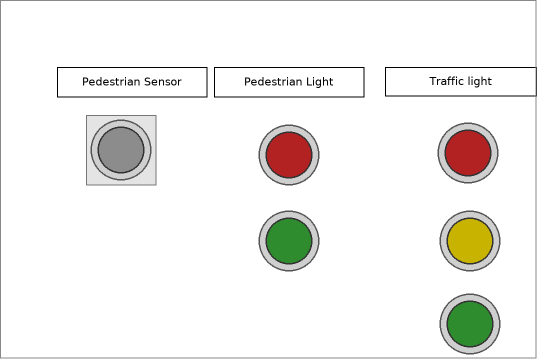
VISUALIZATION Visualization_Trafficlight  // 537x359
    Lamp1 (433,118 70x70), variable: GVL.CarLightRed, style: Lamp-Lamp1-Red
    Lamp1 (435,206 70x70), variable: GVL.CarLightYellow, style: Lamp-Lamp1-Yellow
    Lamp1 (435,289 70x70), variable: GVL.CarLightGreen, style: Lamp-Lamp1-Green
    Rectangle (385,67 152x29), "Traffic light"
    Rectangle (57,67 150x30), "Pedestrian Sensor"
    Lamp1 (254,120 70x70), variable: GVL.PedestrianLightRed, style: Lamp-Lamp1-Red
    Lamp1 (254,206 70x70), variable: GVL.PedestrianLightGreen, style: Lamp-Lamp1-Green
    Rectangle (214,67 150x30), "Pedestrian Light"
    PushSwitch (86,115 70x70), variable: GVL.ButtonPedestrian, behaviour: TOGGLE, style: Switch-PushSwitch-Gray
END_VISUALIZATION

(* stored: Version 1.1.0.1, ProductVersion 3.1.4024.12
   Visu Visualization_Trafficlight: Id {4a0da58c-caeb-4321-b1db-9ac83a6d612b} *)
